ABB RobotStudio station: System_20200221-104554.rsstn

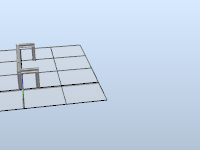
Station Station (saved by RobotStudio 7.0.8728.594)
Layout (positions relative to the parent item):
  - SmartComponent_1 [smart component]
    - PositionSensor [smart component, from Components\PositionSensor.rslib]
        properties: Object=(none); Reference=Global; ReferenceObject=(none); Position=[0 0 0]; Orientation=[0 0 0]
    - LinearMover2 [smart component, from Components\LinearMover2.rslib]
        properties: Object=(none); Direction=[1 0 0]; Distance=0; Duration=0; Reference=Global; ReferenceObject=(none)
  - Track [part] at (0, 0, 500) mm, rotated rx 90 ry 0 rz 0 deg
  - Cart [part] at (-81.51, 337.69, 0) mm, rotated rx 90 ry 0 rz 0 deg
